// TIA Portal project "Metrou_2026" (V15.1)

(* hardware
DEVICE "S71500/ET200MP station_1"  S7-1500 station
   slot 0: "Rail_0"  Rack  6ES7 590-1***0-0AA0
   slot 1: "PLC_1(Scari)"  CPU 1513-1 PN  6ES7 513-1AL02-0AB0  V2.6
      slot 3: "CPU display_1"  6ES7591-1AA00-0AA0
DEVICE "S71500/ET200MP station_2"  S7-1500 station
   slot 0: "Rail_0"  Rack  6ES7 590-1***0-0AA0
   slot 1: "PLC_1(Metrou)"  CPU 1513-1 PN  6ES7 513-1AL02-0AB0  V2.6
      slot 3: "CPU display_1"  6ES7591-1AA00-0AA0
DEVICE "HMI_1(Scari)"  KTP900 Basic PN
   slot 0: "HMI_1(Scari)"  KTP900 Basic PN  6AV2 123-2JB03-0AX0  15.1.0.0
   slot 1: "HMI_RT_1"  KTP900 Basic PN  6AV2 123-2JB03-0AX0  15.1.0.0
   slot 5: "HMI_1(Scari).IE_CP_1"  PROFINET Interface  15.0.1.0
      slot 1: "PROFINET Interface_1"  PROFINET Interface
         slot 1: "Port_1"  Port
DEVICE "HMI_1(Metrou)"  KTP900 Basic PN
   slot 0: "HMI_1(Metrou)"  KTP900 Basic PN  6AV2 123-2JB03-0AX0  15.1.0.0
   slot 1: "HMI_RT_2"  KTP900 Basic PN  6AV2 123-2JB03-0AX0  15.1.0.0
   slot 5: "HMI_1(Metrou).IE_CP_1"  PROFINET Interface  15.0.1.0
      slot 1: "PROFINET Interface_1"  PROFINET Interface
         slot 1: "Port_1"  Port
*)

// ===== PLC "PLC_1(Scari)"  CPU 1513-1 PN =====

// folder: Alarme/Avarii

DATA_BLOCK "Alarme"   // DB1
{ S7_Optimized_Access := 'TRUE' }
VERSION : 0.1
   VAR
      gather : Word;
      "array" : Array[0..15] of Bool;
   END_VAR
BEGIN
END_DATA_BLOCK

DATA_BLOCK "Avarii"   // DB2
{ S7_Optimized_Access := 'TRUE' }
VERSION : 0.1
   VAR
      esd : Bool;
      btn_esd : Bool;
      reset_esd : Bool;
      avarie_1 : Bool;
      avarie_2 : Bool;
      avarie_3 : Bool;
      avarie_4 : Bool;
      btn_avarie_1 : Bool;
      btn_avarie_2 : Bool;
      btn_avarie_3 : Bool;
      btn_avarie_4 : Bool;
      reset_avarie_1 : Bool;
      reset_avarie_2 : Bool;
      reset_avarie_3 : Bool;
      reset_avarie_4 : Bool;
   END_VAR
BEGIN
END_DATA_BLOCK

// folder: Instante_FB

DATA_BLOCK "ESD_Instanta"   // DB4
{ S7_Optimized_Access := 'TRUE' }
VERSION : 0.1
// stored: InstanceOfName Avarei/ESD_FB
"Avarei/ESD_FB"
BEGIN
END_DATA_BLOCK

DATA_BLOCK "Scara1_Instanta_Alarme"   // DB5
{ S7_Optimized_Access := 'TRUE' }
VERSION : 0.1
// stored: InstanceOfName Avarei/ESD_FB
"Avarei/ESD_FB"
BEGIN
END_DATA_BLOCK

DATA_BLOCK "Scara2_Instanta_Alarme"   // DB6
{ S7_Optimized_Access := 'TRUE' }
VERSION : 0.1
// stored: InstanceOfName Avarei/ESD_FB
"Avarei/ESD_FB"
BEGIN
END_DATA_BLOCK

DATA_BLOCK "Scara3_Instanta_Alarme"   // DB7
{ S7_Optimized_Access := 'TRUE' }
VERSION : 0.1
// stored: InstanceOfName Avarei/ESD_FB
"Avarei/ESD_FB"
BEGIN
END_DATA_BLOCK

DATA_BLOCK "Scara4_Instanta_Alarme"   // DB8
{ S7_Optimized_Access := 'TRUE' }
VERSION : 0.1
// stored: InstanceOfName Avarei/ESD_FB
"Avarei/ESD_FB"
BEGIN
END_DATA_BLOCK

DATA_BLOCK "Scara1_Instanta_FB"   // DB9
{ S7_Optimized_Access := 'TRUE' }
VERSION : 0.1
// stored: InstanceOfName Scari
"Scari"
BEGIN
END_DATA_BLOCK

// folder: Scari

DATA_BLOCK "Scara1_DB"   // DB3
{ S7_Optimized_Access := 'TRUE' }
VERSION : 0.1
   VAR
      "mod" : DInt;
      btn_start : Bool;
      btn_stop : Bool;
      senzor_persoana_urcare : Bool;
      senzor_persoana_coborare : Bool;
      stea_urcare : Bool;
      stea_coborare : Bool;
      triunghi_urcare : Bool;
      triunghi_coborare : Bool;
      et_stea_u : Time;
      et_stea_c : Time;
      et_persoana_u : Time;
      et_persoana_c : Time;
   END_VAR
BEGIN
END_DATA_BLOCK

// folder: (top level)

ORGANIZATION_BLOCK "Main"   // OB1, LAD, ProgramCycle
TITLE = "Main Program Sweep (Cycle)"
{ S7_Optimized_Access := 'TRUE' }
VERSION : 0.1
   VAR_INPUT
      Initial_Call : Bool;   // Initial call of this OB
      Remanence : Bool;   // =True, if remanent data are available
   END_VAR
BEGIN

REGION Network 1: gather de alarme
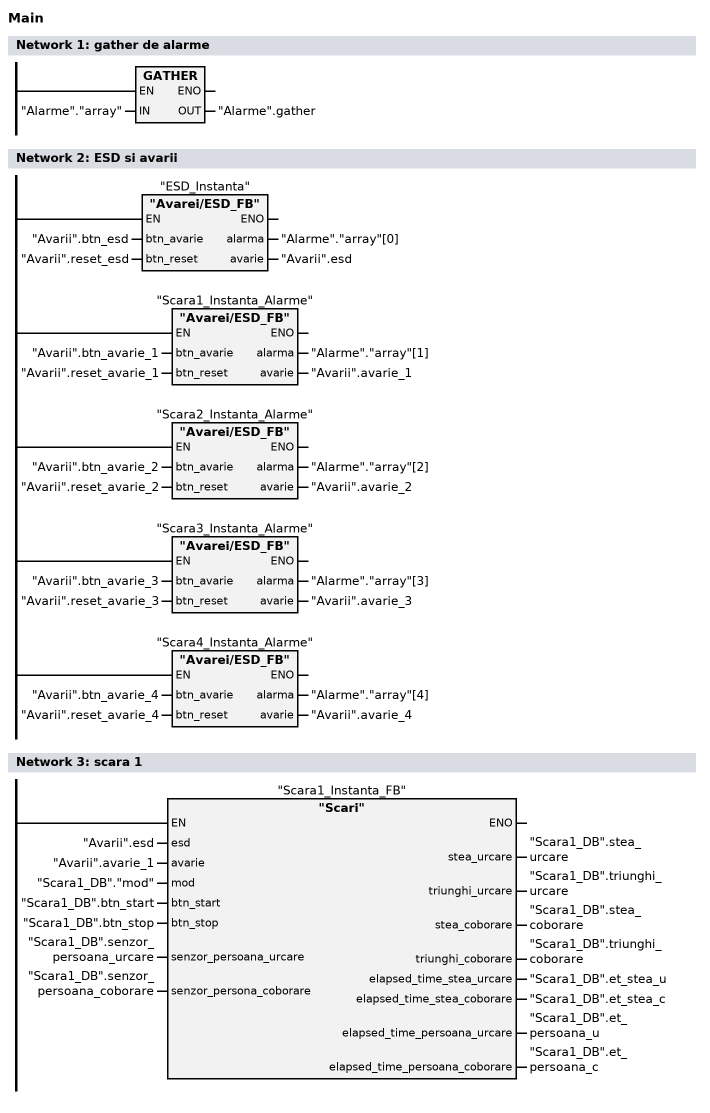
   GATHER(IN := "Alarme"."array", OUT => "Alarme".gather);
END_REGION

REGION Network 2: ESD si avarii
   RUNG wire#powerrail
      "ESD_Instanta"(btn_avarie := "Avarii".btn_esd, btn_reset := "Avarii".reset_esd, alarma => "Alarme"."array"[0], avarie => "Avarii".esd)
   END_RUNG
   RUNG wire#powerrail
      "Scara1_Instanta_Alarme"(btn_avarie := "Avarii".btn_avarie_1, btn_reset := "Avarii".reset_avarie_1, alarma => "Alarme"."array"[1], avarie => "Avarii".avarie_1)
   END_RUNG
   RUNG wire#powerrail
      "Scara2_Instanta_Alarme"(btn_avarie := "Avarii".btn_avarie_2, btn_reset := "Avarii".reset_avarie_2, alarma => "Alarme"."array"[2], avarie => "Avarii".avarie_2)
   END_RUNG
   RUNG wire#powerrail
      "Scara3_Instanta_Alarme"(btn_avarie := "Avarii".btn_avarie_3, btn_reset := "Avarii".reset_avarie_3, alarma => "Alarme"."array"[3], avarie => "Avarii".avarie_3)
   END_RUNG
   RUNG wire#powerrail
      "Scara4_Instanta_Alarme"(btn_avarie := "Avarii".btn_avarie_4, btn_reset := "Avarii".reset_avarie_4, alarma => "Alarme"."array"[4], avarie => "Avarii".avarie_4)
   END_RUNG
   // the same network as SCL:
   "ESD_Instanta"(btn_avarie := "Avarii".btn_esd,   // "Avarei/ESD_FB"
                  btn_reset := "Avarii".reset_esd,
                  alarma => "Alarme"."array"[0],
                  avarie => "Avarii".esd);
   "Scara1_Instanta_Alarme"(btn_avarie := "Avarii".btn_avarie_1,   // "Avarei/ESD_FB"
                           btn_reset := "Avarii".reset_avarie_1,
                           alarma => "Alarme"."array"[1],
                           avarie => "Avarii".avarie_1);
   "Scara2_Instanta_Alarme"(btn_avarie := "Avarii".btn_avarie_2,   // "Avarei/ESD_FB"
                           btn_reset := "Avarii".reset_avarie_2,
                           alarma => "Alarme"."array"[2],
                           avarie => "Avarii".avarie_2);
   "Scara3_Instanta_Alarme"(btn_avarie := "Avarii".btn_avarie_3,   // "Avarei/ESD_FB"
                           btn_reset := "Avarii".reset_avarie_3,
                           alarma => "Alarme"."array"[3],
                           avarie => "Avarii".avarie_3);
   "Scara4_Instanta_Alarme"(btn_avarie := "Avarii".btn_avarie_4,   // "Avarei/ESD_FB"
                           btn_reset := "Avarii".reset_avarie_4,
                           alarma => "Alarme"."array"[4],
                           avarie => "Avarii".avarie_4);
END_REGION

REGION Network 3: scara 1
   RUNG wire#powerrail
      "Scara1_Instanta_FB"(esd := "Avarii".esd, avarie := "Avarii".avarie_1, "mod" := "Scara1_DB"."mod", btn_start := "Scara1_DB".btn_start, btn_stop := "Scara1_DB".btn_stop, senzor_persoana_urcare := "Scara1_DB".senzor_persoana_urcare, senzor_persona_coborare := "Scara1_DB".senzor_persoana_coborare, stea_urcare => "Scara1_DB".stea_urcare, triunghi_urcare => "Scara1_DB".triunghi_urcare, stea_coborare => "Scara1_DB".stea_coborare, triunghi_coborare => "Scara1_DB".triunghi_coborare, elapsed_time_stea_urcare => "Scara1_DB".et_stea_u, elapsed_time_stea_coborare => "Scara1_DB".et_stea_c, elapsed_time_persoana_urcare => "Scara1_DB".et_persoana_u, elapsed_time_persoana_coborare => "Scara1_DB".et_persoana_c)
   END_RUNG
   // the same network as SCL:
   "Scara1_Instanta_FB"(esd := "Avarii".esd,   // "Scari"
                        avarie := "Avarii".avarie_1,
                        "mod" := "Scara1_DB"."mod",
                        btn_start := "Scara1_DB".btn_start,
                        btn_stop := "Scara1_DB".btn_stop,
                        senzor_persoana_urcare := "Scara1_DB".senzor_persoana_urcare,
                        senzor_persona_coborare := "Scara1_DB".senzor_persoana_coborare,
                        stea_urcare => "Scara1_DB".stea_urcare,
                        triunghi_urcare => "Scara1_DB".triunghi_urcare,
                        stea_coborare => "Scara1_DB".stea_coborare,
                        triunghi_coborare => "Scara1_DB".triunghi_coborare,
                        elapsed_time_stea_urcare => "Scara1_DB".et_stea_u,
                        elapsed_time_stea_coborare => "Scara1_DB".et_stea_c,
                        elapsed_time_persoana_urcare => "Scara1_DB".et_persoana_u,
                        elapsed_time_persoana_coborare => "Scara1_DB".et_persoana_c);
END_REGION
END_ORGANIZATION_BLOCK

// folder: Alarme/Avarii

FUNCTION_BLOCK "Avarei/ESD_FB"   // FB2, LAD
{ S7_Optimized_Access := 'TRUE' }
VERSION : 0.1
   VAR_OUTPUT
      alarma : Bool;
      avarie : Bool;
   END_VAR
   VAR_IN_OUT
      btn_avarie : Bool;
      btn_reset : Bool;
   END_VAR
   VAR
      ton : TON_TIME;
   END_VAR
BEGIN

REGION Network 1: seteaza avaria
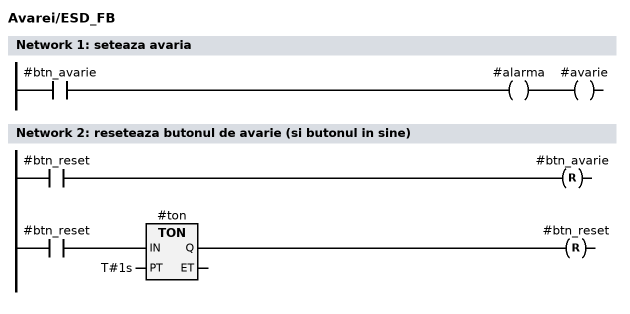
   RUNG wire#powerrail
      Contact( #btn_avarie )
      Coil( #alarma )
      Coil( #avarie )
   END_RUNG
   // the same network as SCL:
   #alarma := #btn_avarie;
   #avarie := #btn_avarie;
END_REGION

REGION Network 2: reseteaza butonul de avarie (si butonul in sine)
   IF #btn_reset THEN #btn_avarie := FALSE; END_IF;
   #ton(IN := #btn_reset, PT := T#1s);   // TON
   IF #ton.Q THEN #btn_reset := FALSE; END_IF;
END_REGION
END_FUNCTION_BLOCK

// folder: Scari

FUNCTION_BLOCK "Scari"   // FB1, LAD
{ S7_Optimized_Access := 'TRUE' }
VERSION : 0.1
   VAR_INPUT
      esd : Bool;
      avarie : Bool;
      "mod" : DInt;
   END_VAR
   VAR_OUTPUT
      stea_urcare : Bool;
      triunghi_urcare : Bool;
      stea_coborare : Bool;
      triunghi_coborare : Bool;
      elapsed_time_stea_urcare : Time;
      elapsed_time_stea_coborare : Time;
      elapsed_time_persoana_urcare : Time;
      elapsed_time_persoana_coborare : Time;
   END_VAR
   VAR_IN_OUT
      btn_start : Bool;
      btn_stop : Bool;
      senzor_persoana_urcare : Bool;
      senzor_persona_coborare : Bool;
   END_VAR
   VAR
      ton_stea_urcare : TON_TIME;
      ton_stea_coborare : TON_TIME;
      ton_persoana_urcare : TON_TIME;
      ton_persoana_coborare : TON_TIME;
      ton_btn_stop : TON_TIME;
      permisiune_urcare : Bool;
      permisiune_coborare : Bool;
      plecare_stea_urcare : Bool;
      plecare_stea_coborare : Bool;
      plecare_triunghi_urcare : Bool;
      plecare_triunghi_coborare : Bool;
      terminat_timer_stea_urcare : Bool;
      terminat_timer_stea_coborare : Bool;
      terminat_persoana_urcare : Bool;
      terminat_persoana_coborare : Bool;
   END_VAR
BEGIN

REGION Network 1: Reseteaza senzorii daca modul nu este setat
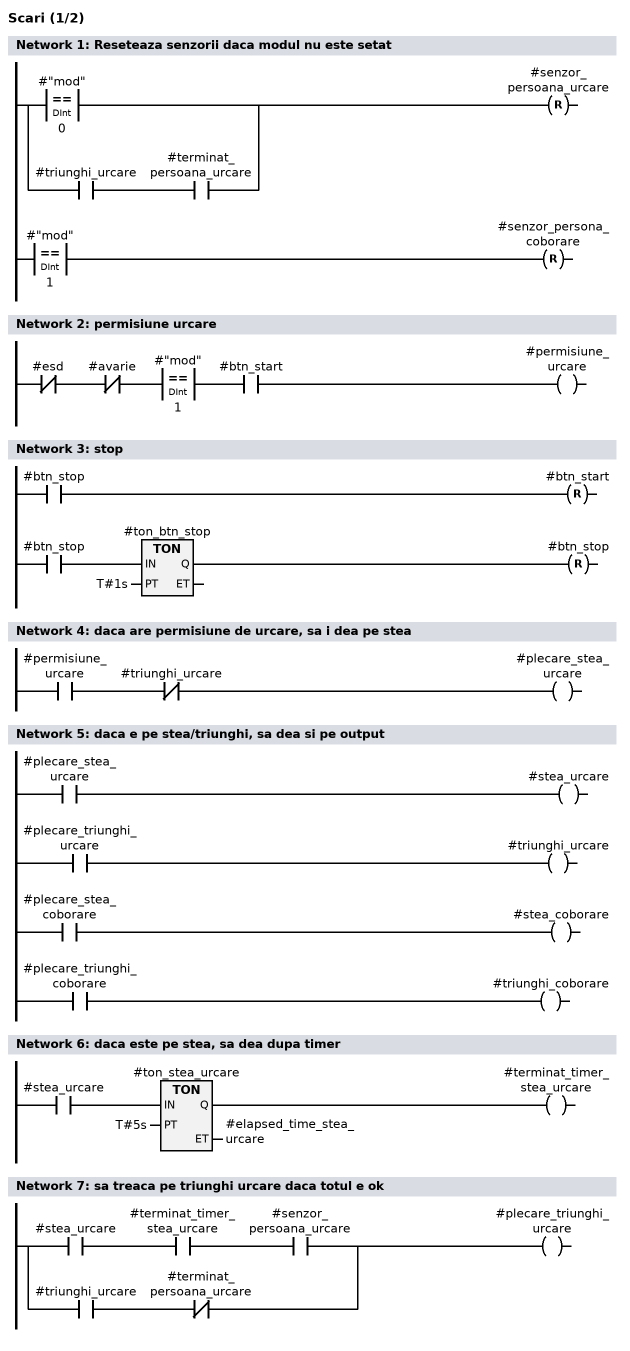
   RUNG wire#powerrail
      { S7_Templates := "SrcType := DInt" } EQ_Contact(in1 := #"mod", in2 := 0)
      wire#w1
      R_Coil( #senzor_persoana_urcare )
   END_RUNG
   RUNG wire#powerrail
      Contact( #triunghi_urcare )
      Contact( #terminat_persoana_urcare )
   END_RUNG wire#w1
   RUNG wire#powerrail
      { S7_Templates := "SrcType := DInt" } EQ_Contact(in1 := #"mod", in2 := 1)
      R_Coil( #senzor_persona_coborare )
   END_RUNG
   // the same network as SCL:
   IF (#"mod" = 0) OR (#triunghi_urcare AND #terminat_persoana_urcare) THEN
       #senzor_persoana_urcare := FALSE;
   END_IF;
   IF #"mod" = 1 THEN #senzor_persona_coborare := FALSE; END_IF;
END_REGION

REGION Network 2: permisiune urcare
   RUNG wire#powerrail
      I_Contact( #esd )
      I_Contact( #avarie )
      { S7_Templates := "SrcType := DInt" } EQ_Contact(in1 := #"mod", in2 := 1)
      Contact( #btn_start )
      Coil( #permisiune_urcare )
   END_RUNG
   // the same network as SCL:
   #permisiune_urcare := NOT #esd AND NOT #avarie AND (#"mod" = 1) AND #btn_start;
END_REGION

REGION Network 3: stop
   IF #btn_stop THEN #btn_start := FALSE; END_IF;
   #ton_btn_stop(IN := #btn_stop, PT := T#1s);   // TON
   IF #ton_btn_stop.Q THEN #btn_stop := FALSE; END_IF;
END_REGION

REGION Network 4: daca are permisiune de urcare, sa i dea pe stea
   RUNG wire#powerrail
      Contact( #permisiune_urcare )
      I_Contact( #triunghi_urcare )
      Coil( #plecare_stea_urcare )
   END_RUNG
   // the same network as SCL:
   #plecare_stea_urcare := #permisiune_urcare AND NOT #triunghi_urcare;
END_REGION

REGION Network 5: daca e pe stea/triunghi, sa dea si pe output
   RUNG wire#powerrail
      Contact( #plecare_stea_urcare )
      Coil( #stea_urcare )
   END_RUNG
   RUNG wire#powerrail
      Contact( #plecare_triunghi_urcare )
      Coil( #triunghi_urcare )
   END_RUNG
   RUNG wire#powerrail
      Contact( #plecare_stea_coborare )
      Coil( #stea_coborare )
   END_RUNG
   RUNG wire#powerrail
      Contact( #plecare_triunghi_coborare )
      Coil( #triunghi_coborare )
   END_RUNG
   // the same network as SCL:
   #stea_urcare := #plecare_stea_urcare;
   #triunghi_urcare := #plecare_triunghi_urcare;
   #stea_coborare := #plecare_stea_coborare;
   #triunghi_coborare := #plecare_triunghi_coborare;
END_REGION

REGION Network 6: daca este pe stea, sa dea dupa timer
   #ton_stea_urcare(IN := #stea_urcare, PT := T#5s, ET => #elapsed_time_stea_urcare);   // TON
   #terminat_timer_stea_urcare := #ton_stea_urcare.Q;
END_REGION

REGION Network 7: sa treaca pe triunghi urcare daca totul e ok
   RUNG wire#powerrail
      Contact( #stea_urcare )
      Contact( #terminat_timer_stea_urcare )
      Contact( #senzor_persoana_urcare )
      wire#w1
      Coil( #plecare_triunghi_urcare )
   END_RUNG
   RUNG wire#powerrail
      Contact( #triunghi_urcare )
      I_Contact( #terminat_persoana_urcare )
   END_RUNG wire#w1
   // the same network as SCL:
   #plecare_triunghi_urcare := (#stea_urcare AND #terminat_timer_stea_urcare AND #senzor_persoana_urcare) OR (#triunghi_urcare AND NOT #terminat_persoana_urcare);
END_REGION

REGION Network 8: daca simte persoana pe urcare, sa i dea un timer de 15s pana trece iar la stea
   // timpul este hardcodat pe baza la lungimea scarii si timpul cat ii ia sa parcurga lungimea cu o persoana
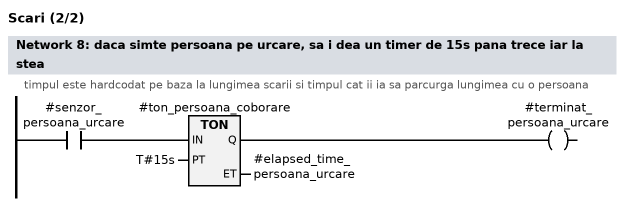
   #ton_persoana_coborare(IN := #senzor_persoana_urcare, PT := T#15s, ET => #elapsed_time_persoana_urcare);   // TON
   #terminat_persoana_urcare := #ton_persoana_coborare.Q;
END_REGION
END_FUNCTION_BLOCK

// ===== PLC "PLC_1(Metrou)"  CPU 1513-1 PN =====

ORGANIZATION_BLOCK "Main"   // OB1, LAD, ProgramCycle
TITLE = "Main Program Sweep (Cycle)"
{ S7_Optimized_Access := 'TRUE' }
VERSION : 0.1
   VAR_INPUT
      Initial_Call : Bool;   // Initial call of this OB
      Remanence : Bool;   // =True, if remanent data are available
   END_VAR
BEGIN
END_ORGANIZATION_BLOCK

(* ===== HMI "HMI_RT_1" =====
connection "HMI_Connection_1": ETHERNET, SMART_S7_1500_OMS

HMI tags "Default tag table"
   "Alarme_gather" : Word = PLC Alarme.gather, 1 s

discrete alarms
   1: 'ESD', class Errors, trigger "Alarme_gather" bit 0
   2: 'Avarie la scara 1', class Errors, trigger "Alarme_gather" bit 1
   3: 'Avarie la scara 2', class Errors, trigger "Alarme_gather" bit 2
   4: 'Avarie la scara 3', class Errors, trigger "Alarme_gather" bit 3
   5: 'Avarie la scara 4', class Errors, trigger "Alarme_gather" bit 4
*)

(* ===== HMI "HMI_RT_2" =====

Template "Template_1" 800x480
   Button "Template_Button" at 722,440 size 55x39; TextOff 'Text'
   Button "Template_Button_1" at 622,440 size 55x39; TextOff 'Text'
   Button "Template_Button_2" at 522,440 size 55x39; TextOff 'Text'
   Button "Template_Button_3" at 422,440 size 55x39; TextOff 'Text'
   Button "Template_Button_4" at 322,440 size 55x39; TextOff 'Text'
   Button "Template_Button_5" at 222,440 size 55x39; TextOff 'Text'
   Button "Template_Button_6" at 122,440 size 55x39; TextOff 'Text'
   Button "Template_Button_7" at 22,440 size 55x39; TextOff 'Text'

screen "Main" 800x480, template "Template_1"
   TextField "HmiScreenItemData" at 80,206 size 640x22; Text 'Welcome to HMI_1 (KTP900 Basic+ PN)!'
*)